(* 	Disclaimer
	All sample code provided by Beckhoff Automation LLC are for illustrative purposes only and are provided “as is” and without any warranties, express or implied.
	Actual implementations in applications will vary significantly.
	Beckhoff Automation LLC shall have no liability for, and does not waive any rights in relation to, any code samples that it provides or the use of such code samples for any purpose.
*)
FUNCTION_BLOCK FB_Actuator
VAR_INPUT
	Activate: BOOL;
	Deactivate: BOOL;
	EDM_Activated: BOOL;
	EDM_Deactivated: BOOL;
	ErrAck: BOOL;
	TimeOn: TIME := T#2S;
	TimeOff: TIME := T#2S;
END_VAR
VAR_OUTPUT
	Activated: BOOL;
	Busy: BOOL;
	Error: BOOL;
	ErrorId: UDINT;
END_VAR
VAR
	eState :(eInit, eIdle, eActivate, eDeactivate, eError);
	tonWD_On: TON;
	tonWD_Off: TON;
END_VAR

// Activating Watchdog
tonWD_On.IN := Activated AND NOT EDM_Activated;
tonWD_On.PT := TimeOn;
IF tonWD_On.Q THEN
	Error := TRUE;
	ErrorId := 1;
END_IF

// Deactivating Watchdog
tonWD_Off.IN := NOT Activated AND NOT EDM_Deactivated;
tonWD_Off.PT := TimeOff;
IF tonWD_Off.Q THEN
	Error := TRUE;
	ErrorId := 2;
END_IF

// State Machine
CASE eState OF
	eInit:
		Activated := FALSE;
		Busy := FALSE;
		Error := FALSE;
		ErrorId := 0;
		eState := eIdle;
	
	eIdle:
		Busy := FALSE;
		IF NOT Activated AND Activate THEN
			eState := eActivate;
		ELSIF Activated AND Deactivate THEN
			eState := eDeactivate;
		END_IF
		
	eActivate:
		Busy := TRUE;
		Activated := TRUE;
		IF NOT Activate OR EDM_Activated THEN
			eState := eIdle;
		END_IF
	
	eDeactivate:
		Busy := TRUE;
		Activated := FALSE;
		IF Activate OR EDM_Deactivated THEN
			eState := eIdle;
		END_IF	
		
	eError:
		IF ErrAck THEN
			eState := eInit;
		END_IF
	
END_CASE

// Call function blocks
tonWD_On();
tonWD_Off();

END_FUNCTION_BLOCK

(* stored: Version 1.1.0.1, ProductVersion 3.1.4024.12
   POU FB_Actuator: Id {a96b305c-5f90-49ef-90b2-631d225a4db4}, SpecialFunc None *)
